PROGRAM P_Demo_FB_DMXSendRDMCommand
VAR
    fbSendRdm         : FB_DMXSendRDMCommand;         // 通用 RDM 命令发送
    stDmxCmdBuffer    : ST_DMXCommandBuffer;          // 与通讯 FB 共用
    wTargetManufId    : WORD := 16#4241;              // 目标灯具厂商 ID
    dwTargetDeviceId  : DWORD := 16#12131415;         // 目标灯具设备 ID
    byTargetPort      : BYTE := 0;                    // 根设备通道 0
    wTargetSubDevice  : WORD := 0;                    // 0 = 根设备
    eCmdClass         : E_DMXCommandClass;            // GET / SET ...
    eParamId          : E_DMXParameterId;             // 目标 PID
    byParamLen        : BYTE := 0;                    // 参数数据长度
    arrParamData      : ARRAY [0..255] OF BYTE;       // 参数数据
    bDoSend           : BOOL := FALSE;                // 在线给一次上升沿触发
    bBusy             : BOOL;
    bError            : BOOL;
    udiErrId          : UDINT;
    byRespMsgCount    : BYTE;                         // 设备排队消息数
    byRespLen         : BYTE;                         // 应答字节数
    arrRespData       : ARRAY [0..255] OF BYTE;       // 应答数据
END_VAR

// ============================================================
// Tc2_DMX.FB_DMXSendRDMCommand 演示程序
// ============================================================
// 场景：某灯具支持厂商自定义 PID，库里没有专用 FB，需手工构造 RDM 命令读取。
// 价值：按 RDM 标准填 CC/PID/参数即可发任意命令取回原始应答，覆盖全部 RDM 能力，无需等专用 FB。
// 验证：设好 eCmdClass / eParamId / arrParamData 后给 bDoSend 一次上升沿 -> bBusy 短暂 TRUE -> 回 FALSE 后 arrRespData[0..byRespLen-1] 是应答；用 GET 一个标准 PID（如 DEVICE_INFO）先验证链路。
// 验证步骤：
//   1. 右键 PLC 项目下 POUs 文件夹 → Add → Existing Item → 选本 .TcPOU 文件
//   2. 引用 Tc2_DMX；同项目里放一个 FB_EL6851CommunicationEx 实例并共用 stDmxCmdBuffer（非 CycleMode）
//   3. 编译 → 登录 → 运行；按上方『验证』行在线给上升沿观察
// ============================================================

eCmdClass := eDMXCommandClassGetCommand;     // 示例：GET 命令
eParamId  := eDMXParameterIdDeviceInfo;      // 示例：读 DEVICE_INFO（标准 PID）
byParamLen := 0;                             // GET DEVICE_INFO 无参数数据

fbSendRdm(
    bStart                     := bDoSend,
    wDestinationManufacturerId := wTargetManufId,
    dwDestinationDeviceId      := dwTargetDeviceId,
    byPortId                   := byTargetPort,
    wSubDevice                 := wTargetSubDevice,
    eCommandClass              := eCmdClass,
    eParameterId               := eParamId,
    byParameterDataLength      := byParamLen,
    arrParameterData           := arrParamData,
    dwOptions                  := 0,
    stCommandBuffer            := stDmxCmdBuffer,
    bBusy                      => bBusy,
    bError                     => bError,
    udiErrorId                 => udiErrId,
    byResponseMessageCount     => byRespMsgCount,
    byResponseDataLength       => byRespLen,
    arrResponseData            => arrRespData
);

END_PROGRAM

(* stored: Version 1.1.0.1, ProductVersion 3.1.4024.5
   POU P_Demo_FB_DMXSendRDMCommand: Id {bc0a4ef2-08cc-5028-bb1e-33ca19b0fcb1}, SpecialFunc None *)
